// TIA Portal V18 export
ORGANIZATION_BLOCK "14-WireDraw"   // OB125, LAD, ProgramCycle
TITLE = "Main Program Sweep (Cycle)"
{ S7_Optimized_Access := 'TRUE' }
VERSION : 0.1
// stored: AutoNumber true, IsIECCheckEnabled false, SetENOAutomatically false
   VAR_INPUT
      Initial_Call : Bool;   // Initial call of this OB
      Remanence : Bool;   // =True, if remanent data are available
   END_VAR
   VAR_TEMP
      "Temp_1 (NormScale) Wire" : Real;
      "Temp_2 (NormScale) Inclanation" : Real;
      Temp_3 : Real;
      "Temp_4 (Radyan)" : Real;
      Temp_5 : Real;
   END_VAR
BEGIN

REGION Network 1: WireDraw Encoder _ Height Real
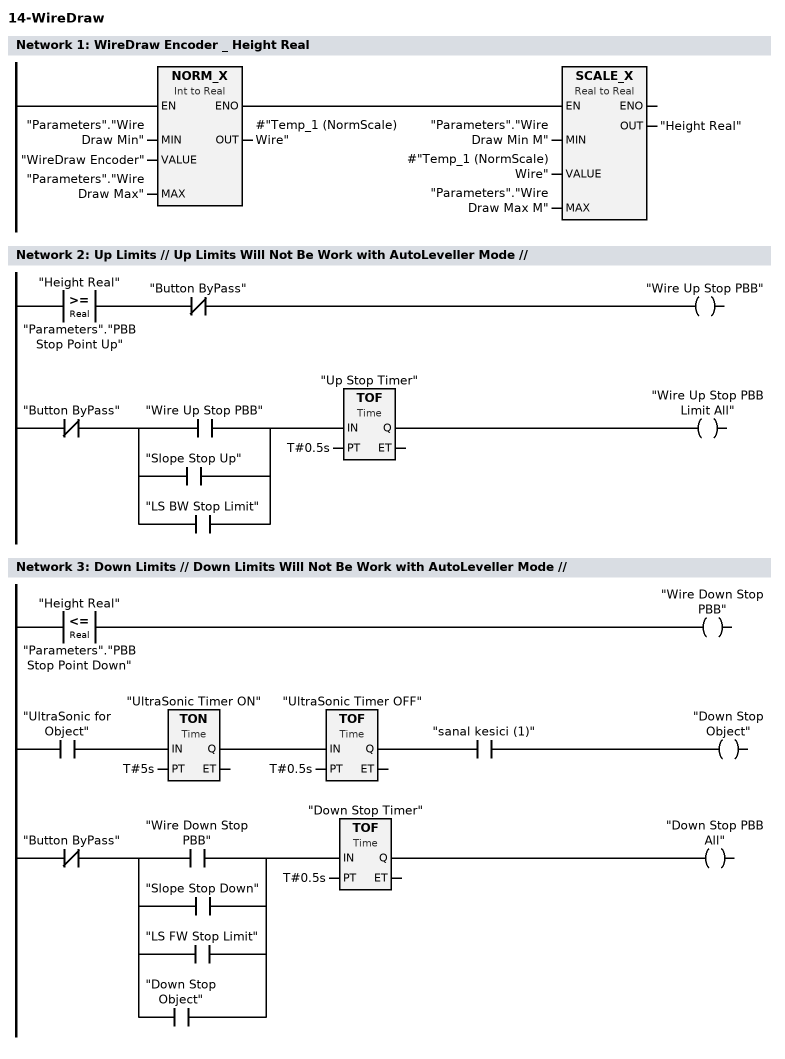
   RUNG wire#powerrail
      { S7_Templates := "[SrcType := Int, DestType := Real]" } Normalize(min := "Parameters"."Wire Draw Min", value := "WireDraw Encoder", max := "Parameters"."Wire Draw Max", out => #"Temp_1 (NormScale) Wire")
      { S7_Templates := "[SrcType := Real, DestType := Real]" } Scale(min := "Parameters"."Wire Draw Min M", value := #"Temp_1 (NormScale) Wire", max := "Parameters"."Wire Draw Max M", out => "Height Real")
   END_RUNG
   // the same network as SCL:
   #"Temp_1 (NormScale) Wire" := NORM_X(MIN := "Parameters"."Wire Draw Min", VALUE := "WireDraw Encoder", MAX := "Parameters"."Wire Draw Max");
   "Height Real" := SCALE_X(MIN := "Parameters"."Wire Draw Min M", VALUE := #"Temp_1 (NormScale) Wire", MAX := "Parameters"."Wire Draw Max M");
END_REGION

REGION Network 2: Up Limits // Up Limits Will Not Be Work with AutoLeveller Mode //
   RUNG wire#powerrail
      { S7_Templates := "SrcType := Real" } GE_Contact(in1 := "Height Real", in2 := "Parameters"."PBB Stop Point Up")
      I_Contact( "Button ByPass" )
      Coil( "Wire Up Stop PBB" )
   END_RUNG
   RUNG wire#powerrail
      I_Contact( "Button ByPass" )
      wire#w1
      Contact( "Wire Up Stop PBB" )
      wire#w2
      { S7_Templates := "time_type := Time" } "Up Stop Timer".TOF(pt := T#0.5s, et =>)
      Coil( "Wire Up Stop PBB Limit All" )
   END_RUNG
   RUNG wire#w1
      Contact( "Slope Stop Up" )
   END_RUNG wire#w2
   RUNG wire#w1
      Contact( "LS BW Stop Limit" )
   END_RUNG wire#w2
   // the same network as SCL:
   "Wire Up Stop PBB" := ("Height Real" >= "Parameters"."PBB Stop Point Up") AND NOT "Button ByPass";
   "Up Stop Timer".TOF(IN := NOT "Button ByPass" AND ("Wire Up Stop PBB" OR "Slope Stop Up" OR "LS BW Stop Limit"),
                       PT := T#0.5s);
   "Wire Up Stop PBB Limit All" := "Up Stop Timer".Q;
END_REGION

REGION Network 3: Down Limits // Down Limits Will Not Be Work with AutoLeveller Mode //
   RUNG wire#powerrail
      { S7_Templates := "SrcType := Real" } LE_Contact(in1 := "Height Real", in2 := "Parameters"."PBB Stop Point Down")
      Coil( "Wire Down Stop PBB" )
   END_RUNG
   RUNG wire#powerrail
      Contact( "UltraSonic for Object" )
      { S7_Templates := "time_type := Time" } "UltraSonic Timer ON".TON(pt := T#5s, et =>)
      { S7_Templates := "time_type := Time" } "UltraSonic Timer OFF".TOF(pt := T#0.5s, et =>)
      Contact( "sanal kesici (1)" )
      Coil( "Down Stop Object" )
   END_RUNG
   RUNG wire#powerrail
      I_Contact( "Button ByPass" )
      wire#w1
      Contact( "Wire Down Stop PBB" )
      wire#w2
      { S7_Templates := "time_type := Time" } "Down Stop Timer".TOF(pt := T#0.5s, et =>)
      Coil( "Down Stop PBB All" )
   END_RUNG
   RUNG wire#w1
      Contact( "Slope Stop Down" )
   END_RUNG wire#w2
   RUNG wire#w1
      Contact( "LS FW Stop Limit" )
   END_RUNG wire#w2
   RUNG wire#w1
      Contact( "Down Stop Object" )
   END_RUNG wire#w2
   // the same network as SCL:
   "Wire Down Stop PBB" := "Height Real" <= "Parameters"."PBB Stop Point Down";
   "UltraSonic Timer ON".TON(IN := "UltraSonic for Object", PT := T#5s);
   "UltraSonic Timer OFF".TOF(IN := "UltraSonic Timer ON".Q, PT := T#0.5s);
   "Down Stop Object" := "UltraSonic Timer OFF".Q AND "sanal kesici (1)";
   "Down Stop Timer".TOF(IN := NOT "Button ByPass" AND ("Wire Down Stop PBB" OR "Slope Stop Down" OR "LS FW Stop Limit" OR "Down Stop Object"),
                         PT := T#0.5s);
   "Down Stop PBB All" := "Down Stop Timer".Q;
END_REGION
END_ORGANIZATION_BLOCK
